# EPICS substitutions: psd.substitutions
file "/epics/iocs/bpm-psd/psd.db"
{
pattern
{P                        }
{"SR:C30-APHLA{BPM:1}"    }
{"SR:C30-APHLA{BPM:2}"    }
{"SR:C30-APHLA{BPM:3}"    }
{"SR:C30-APHLA{BPM:4}"    }
{"SR:C30-APHLA{BPM:5}"    }
{"SR:C30-APHLA{BPM:6}"    }
{"SR:C01-APHLA{BPM:1}"    }
{"SR:C01-APHLA{BPM:2}"    }
{"SR:C01-APHLA{BPM:3}"    }
{"SR:C01-APHLA{BPM:4}"    }
{"SR:C01-APHLA{BPM:5}"    }
{"SR:C01-APHLA{BPM:6}"    }
{"SR:C02-APHLA{BPM:1}"    }
{"SR:C02-APHLA{BPM:2}"    }
{"SR:C02-APHLA{BPM:3}"    }
{"SR:C02-APHLA{BPM:4}"    }
{"SR:C02-APHLA{BPM:5}"    }
{"SR:C02-APHLA{BPM:6}"    }
{"SR:C03-APHLA{BPM:1}"    }
{"SR:C03-APHLA{BPM:2}"    }
{"SR:C03-APHLA{BPM:3}"    }
{"SR:C03-APHLA{BPM:4}"    }
{"SR:C03-APHLA{BPM:5}"    }
{"SR:C03-APHLA{BPM:6}"    }
{"SR:C04-APHLA{BPM:1}"    }
{"SR:C04-APHLA{BPM:2}"    }
{"SR:C04-APHLA{BPM:3}"    }
{"SR:C04-APHLA{BPM:4}"    }
{"SR:C04-APHLA{BPM:5}"    }
{"SR:C04-APHLA{BPM:6}"    }
{"SR:C05-APHLA{BPM:1}"    }
{"SR:C05-APHLA{BPM:2}"    }
{"SR:C05-APHLA{BPM:3}"    }
{"SR:C05-APHLA{BPM:4}"    }
{"SR:C05-APHLA{BPM:5}"    }
{"SR:C05-APHLA{BPM:6}"    }
{"SR:C06-APHLA{BPM:1}"    }
{"SR:C06-APHLA{BPM:2}"    }
{"SR:C06-APHLA{BPM:3}"    }
{"SR:C06-APHLA{BPM:4}"    }
{"SR:C06-APHLA{BPM:5}"    }
{"SR:C06-APHLA{BPM:6}"    }
{"SR:C07-APHLA{BPM:1}"    }
{"SR:C07-APHLA{BPM:2}"    }
{"SR:C07-APHLA{BPM:3}"    }
{"SR:C07-APHLA{BPM:4}"    }
{"SR:C07-APHLA{BPM:5}"    }
{"SR:C07-APHLA{BPM:6}"    }
{"SR:C08-APHLA{BPM:1}"    }
{"SR:C08-APHLA{BPM:2}"    }
{"SR:C08-APHLA{BPM:3}"    }
{"SR:C08-APHLA{BPM:4}"    }
{"SR:C08-APHLA{BPM:5}"    }
{"SR:C08-APHLA{BPM:6}"    }
{"SR:C09-APHLA{BPM:1}"    }
{"SR:C09-APHLA{BPM:2}"    }
{"SR:C09-APHLA{BPM:3}"    }
{"SR:C09-APHLA{BPM:4}"    }
{"SR:C09-APHLA{BPM:5}"    }
{"SR:C09-APHLA{BPM:6}"    }
{"SR:C10-APHLA{BPM:1}"    }
{"SR:C10-APHLA{BPM:2}"    }
{"SR:C10-APHLA{BPM:3}"    }
{"SR:C10-APHLA{BPM:4}"    }
{"SR:C10-APHLA{BPM:5}"    }
{"SR:C10-APHLA{BPM:6}"    }
{"SR:C11-APHLA{BPM:1}"    }
{"SR:C11-APHLA{BPM:2}"    }
{"SR:C11-APHLA{BPM:3}"    }
{"SR:C11-APHLA{BPM:4}"    }
{"SR:C11-APHLA{BPM:5}"    }
{"SR:C11-APHLA{BPM:6}"    }
{"SR:C12-APHLA{BPM:1}"    }
{"SR:C12-APHLA{BPM:2}"    }
{"SR:C12-APHLA{BPM:3}"    }
{"SR:C12-APHLA{BPM:4}"    }
{"SR:C12-APHLA{BPM:5}"    }
{"SR:C12-APHLA{BPM:6}"    }
{"SR:C13-APHLA{BPM:1}"    }
{"SR:C13-APHLA{BPM:2}"    }
{"SR:C13-APHLA{BPM:3}"    }
{"SR:C13-APHLA{BPM:4}"    }
{"SR:C13-APHLA{BPM:5}"    }
{"SR:C13-APHLA{BPM:6}"    }
{"SR:C14-APHLA{BPM:1}"    }
{"SR:C14-APHLA{BPM:2}"    }
{"SR:C14-APHLA{BPM:3}"    }
{"SR:C14-APHLA{BPM:4}"    }
{"SR:C14-APHLA{BPM:5}"    }
{"SR:C14-APHLA{BPM:6}"    }
{"SR:C15-APHLA{BPM:1}"    }
{"SR:C15-APHLA{BPM:2}"    }
{"SR:C15-APHLA{BPM:3}"    }
{"SR:C15-APHLA{BPM:4}"    }
{"SR:C15-APHLA{BPM:5}"    }
{"SR:C15-APHLA{BPM:6}"    }
{"SR:C16-APHLA{BPM:1}"    }
{"SR:C16-APHLA{BPM:2}"    }
{"SR:C16-APHLA{BPM:3}"    }
{"SR:C16-APHLA{BPM:4}"    }
{"SR:C16-APHLA{BPM:5}"    }
{"SR:C16-APHLA{BPM:6}"    }
{"SR:C17-APHLA{BPM:1}"    }
{"SR:C17-APHLA{BPM:2}"    }
{"SR:C17-APHLA{BPM:3}"    }
{"SR:C17-APHLA{BPM:4}"    }
{"SR:C17-APHLA{BPM:5}"    }
{"SR:C17-APHLA{BPM:6}"    }
{"SR:C18-APHLA{BPM:1}"    }
{"SR:C18-APHLA{BPM:2}"    }
{"SR:C18-APHLA{BPM:3}"    }
{"SR:C18-APHLA{BPM:4}"    }
{"SR:C18-APHLA{BPM:5}"    }
{"SR:C18-APHLA{BPM:6}"    }
{"SR:C19-APHLA{BPM:1}"    }
{"SR:C19-APHLA{BPM:2}"    }
{"SR:C19-APHLA{BPM:3}"    }
{"SR:C19-APHLA{BPM:4}"    }
{"SR:C19-APHLA{BPM:5}"    }
{"SR:C19-APHLA{BPM:6}"    }
{"SR:C20-APHLA{BPM:1}"    }
{"SR:C20-APHLA{BPM:2}"    }
{"SR:C20-APHLA{BPM:3}"    }
{"SR:C20-APHLA{BPM:4}"    }
{"SR:C20-APHLA{BPM:5}"    }
{"SR:C20-APHLA{BPM:6}"    }
{"SR:C21-APHLA{BPM:1}"    }
{"SR:C21-APHLA{BPM:2}"    }
{"SR:C21-APHLA{BPM:3}"    }
{"SR:C21-APHLA{BPM:4}"    }
{"SR:C21-APHLA{BPM:5}"    }
{"SR:C21-APHLA{BPM:6}"    }
{"SR:C22-APHLA{BPM:1}"    }
{"SR:C22-APHLA{BPM:2}"    }
{"SR:C22-APHLA{BPM:3}"    }
{"SR:C22-APHLA{BPM:4}"    }
{"SR:C22-APHLA{BPM:5}"    }
{"SR:C22-APHLA{BPM:6}"    }
{"SR:C23-APHLA{BPM:1}"    }
{"SR:C23-APHLA{BPM:2}"    }
{"SR:C23-APHLA{BPM:3}"    }
{"SR:C23-APHLA{BPM:4}"    }
{"SR:C23-APHLA{BPM:5}"    }
{"SR:C23-APHLA{BPM:6}"    }
{"SR:C24-APHLA{BPM:1}"    }
{"SR:C24-APHLA{BPM:2}"    }
{"SR:C24-APHLA{BPM:3}"    }
{"SR:C24-APHLA{BPM:4}"    }
{"SR:C24-APHLA{BPM:5}"    }
{"SR:C24-APHLA{BPM:6}"    }
{"SR:C25-APHLA{BPM:1}"    }
{"SR:C25-APHLA{BPM:2}"    }
{"SR:C25-APHLA{BPM:3}"    }
{"SR:C25-APHLA{BPM:4}"    }
{"SR:C25-APHLA{BPM:5}"    }
{"SR:C25-APHLA{BPM:6}"    }
{"SR:C26-APHLA{BPM:1}"    }
{"SR:C26-APHLA{BPM:2}"    }
{"SR:C26-APHLA{BPM:3}"    }
{"SR:C26-APHLA{BPM:4}"    }
{"SR:C26-APHLA{BPM:5}"    }
{"SR:C26-APHLA{BPM:6}"    }
{"SR:C27-APHLA{BPM:1}"    }
{"SR:C27-APHLA{BPM:2}"    }
{"SR:C27-APHLA{BPM:3}"    }
{"SR:C27-APHLA{BPM:4}"    }
{"SR:C27-APHLA{BPM:5}"    }
{"SR:C27-APHLA{BPM:6}"    }
{"SR:C28-APHLA{BPM:1}"    }
{"SR:C28-APHLA{BPM:2}"    }
{"SR:C28-APHLA{BPM:3}"    }
{"SR:C28-APHLA{BPM:4}"    }
{"SR:C28-APHLA{BPM:5}"    }
{"SR:C28-APHLA{BPM:6}"    }
{"SR:C29-APHLA{BPM:1}"    }
{"SR:C29-APHLA{BPM:2}"    }
{"SR:C29-APHLA{BPM:3}"    }
{"SR:C29-APHLA{BPM:4}"    }
{"SR:C29-APHLA{BPM:5}"    }
{"SR:C29-APHLA{BPM:6}"    }
{"SR:C04-APHLA{BPM:7}"    }
{"SR:C04-APHLA{BPM:8}"    }
{"SR:C04-APHLA{BPM:9}"    }
{"SR:C04-APHLA{BPM:10}"    }
{"SR:C07-APHLA{BPM:7}"    }
{"SR:C07-APHLA{BPM:8}"    }
{"SR:C07-APHLA{BPM:9}"    }
{"SR:C07-APHLA{BPM:10}"    }
{"SR:C12-APHLA{BPM:7}"    }
{"SR:C12-APHLA{BPM:8}"    }
{"SR:C12-APHLA{BPM:9}"    }
{"SR:C12-APHLA{BPM:10}"    }
{"SR:C19-APHLA{BPM:7}"    }
{"SR:C19-APHLA{BPM:8}"    }
{"SR:C19-APHLA{BPM:9}"    }
{"SR:C19-APHLA{BPM:10}"    }
{"SR:C02-APHLA{BPM:7}"    }
{"SR:C02-APHLA{BPM:8}"    }
{"SR:C03-APHLA{BPM:7}"    }
{"SR:C03-APHLA{BPM:8}"    }
{"SR:C08-APHLA{BPM:7}"    }
{"SR:C08-APHLA{BPM:8}"    }
{"SR:C10-APHLA{BPM:7}"    }
{"SR:C10-APHLA{BPM:8}"    }
{"SR:C11-APHLA{BPM:7}"    }
{"SR:C11-APHLA{BPM:8}"    }
{"SR:C16-APHLA{BPM:7}"    }
{"SR:C16-APHLA{BPM:8}"    }
{"SR:C18-APHLA{BPM:7}"    }
{"SR:C18-APHLA{BPM:8}"    }
{"SR:C21-APHLA{BPM:7}"    }
{"SR:C21-APHLA{BPM:8}"    }
{"SR:C28-APHLA{BPM:7}"    }
{"SR:C28-APHLA{BPM:8}"    }
{"SR:C05-APHLA{BPM:7}"    }
{"SR:C05-APHLA{BPM:8}"    }
{"SR:C05-APHLA{BPM:9}"    }
{"SR:C17-APHLA{BPM:7}"    }
{"SR:C17-APHLA{BPM:8}"    }
{"SR:C17-APHLA{BPM:9}"    }
{"SR:C23-APHLA{BPM:7}"    }
{"SR:C23-APHLA{BPM:8}"    }
{"SR:C23-APHLA{BPM:9}"    }

}
